{attribute 'qualified_only'}
{attribute 'strict'}
TYPE E_Step :
(
	(* special steps *)
	NoStep := -32767,  // No step   
	Unknown := -32000, // unknown step
	
	(* Not Enabled or Errors*)    
	NeOrError := -990, // Not Enabled or Errors
	
	(*MSF Steps*)
	//main steps
	MainStop 		:= 	10, 		// stop
	MainSensor		:=	20,		// sensor area
	MainPiston		:=	30,		// piston area
	MainPause		:=	40,		// pause
	MainEmergency	:=	50,		// emergency
	MainAcknowledge	:=	60,		// acknowledge
	//sub-steps
	Start			:= 	100,
	Measuring		:= 	110,
	Processing		:= 	120,
	conveyor		:=  130,	// a new piece was placed on the conveyor belt
	waiting			:= 	140,	// attesa
	piston			:=	150		// pistone

);
END_TYPE
//  NoStep = '-32767'
//  Unknown = '-32000'
//  NeOrError = '-990'

(* stored: Version 1.1.0.1, ProductVersion 3.1.4024.12
   EnumerationTextList E_Step: Id {fe3a30d3-1d96-4fc1-b1aa-f734a954498a} *)
